(* PLC project marvel_fem, Institute of Astronomy Onto 0.0.1 *)
(* stored: creationDateTime 2025-01-01T00:00:00.0, modificationDateTime 2025-01-01T00:00:00.0 *)

TYPE FemTemperaturesParts : STRUCT
  {attribute 'TcHmiSymbol.Show'}
  basePlate : SimpleTemperature;  (* FEM base plate temperature in °C *)
  {attribute 'TcHmiSymbol.Show'}
  electronics : SimpleTemperature;  (* FEM base plate temperature in °C *)
  {attribute 'TcHmiSymbol.Show'}
  ambient : SimpleTemperature;  (* FEM base plate temperature in °C *)
  {attribute 'TcHmiSymbol.Show'}
  fork : SimpleTemperature;  (* Telescope fork temperature in °C *)
  {attribute 'TcHmiSymbol.Show'}
  truss : SimpleTemperature;  (* Telescope truss temperature in °C *)
  {attribute 'TcHmiSymbol.Show'}
  spider : SimpleTemperature;  (* Telescope spider temperature in °C *)
  {attribute 'TcHmiSymbol.Show'}
  m1Cell : SimpleTemperature;  (* Telescope m1 cell temperature in °C *)
  {attribute 'TcHmiSymbol.Show'}
  spare : SimpleTemperature;  (* Telescope spare temperature in °C *)
END_STRUCT;
END_TYPE

TYPE FemParts : STRUCT
  {attribute 'TcHmiSymbol.Show'}
  fs : MTS50Axis;  (* The fibre selector stage *)
  {attribute 'TcHmiSymbol.Show'}
  cm : MTS50Axis;  (* The calibration mirror stage *)
  {attribute 'TcHmiSymbol.Show'}
  adc1 : ELL14Stage;  (* The ADC rotation 1 stage *)
  {attribute 'TcHmiSymbol.Show'}
  adc2 : ELL14Stage;  (* The ADC rotation 2 stage *)
  {attribute 'TcHmiSymbol.Show'}
  temp : FemTemperatures;  (* Temperatures measured by the front end *)
  {attribute 'TcHmiSymbol.Show'}
  relayGuideCam : SimpleRelay;  (* Relay to power on/off the guiding camera *)
  {attribute 'TcHmiSymbol.Show'}
  relayAcqCam : SimpleRelay;  (* Relay to power on/off the acquisition camera *)
  {attribute 'TcHmiSymbol.Show'}
  relayAdc : SimpleRelay;  (* Relay to power on/off both ADC controllers *)
  {attribute 'TcHmiSymbol.Show'}
  relayTT : SimpleRelay;  (* Relay to power on/off the Tip Tilt piezo driver *)
  {attribute 'TcHmiSymbol.Show'}
  ledHGF : Led;  (* HGF LED *)
  {attribute 'TcHmiSymbol.Show'}
  ledHSF : Led;  (* HSF LED *)
  {attribute 'TcHmiSymbol.Show'}
  ledUGF : Led;  (* UGF LED *)
  {attribute 'TcHmiSymbol.Show'}
  ledUSF : Led;  (* USF LED *)
  {attribute 'TcHmiSymbol.Show'}
  guideCam : GigECamera;  (* Guiding camera *)
  {attribute 'TcHmiSymbol.Show'}
  fvCam : GigECamera;  (* Fibre View camera *)
END_STRUCT;
END_TYPE

TYPE FemProcesses : STRUCT
  {attribute 'TcHmiSymbol.Show'}
  initialize : Process;  (* Start initializing the FEM *)
END_STRUCT;
END_TYPE

TYPE FemTemperaturesStatuses : STRUCT
  {attribute 'OPC.UA.DA' := '1'}
  {attribute 'OPC.UA.DA.Access' := '1'}
  {attribute 'TcHmiSymbol.Show'}
  health : HealthStatus;  (* Are all temperatures OK? *)
END_STRUCT;
END_TYPE

TYPE FemStatuses : STRUCT
  {attribute 'OPC.UA.DA' := '1'}
  {attribute 'OPC.UA.DA.Access' := '1'}
  {attribute 'TcHmiSymbol.Show'}
  init : InitializationStatus;
  {attribute 'OPC.UA.DA' := '1'}
  {attribute 'OPC.UA.DA.Access' := '1'}
  {attribute 'TcHmiSymbol.Show'}
  health : HealthStatus;
  {attribute 'OPC.UA.DA' := '1'}
  {attribute 'OPC.UA.DA.Access' := '1'}
  {attribute 'TcHmiSymbol.Show'}
  busy : BusyStatus;
END_STRUCT;
END_TYPE

TYPE FemConfig : STRUCT
  {attribute 'TcHmiSymbol.Show'}
  fsSim : BOOL;  (* TRUE if the fibre selector axis is simulated *)
  {attribute 'TcHmiSymbol.Show'}
  cmSim : BOOL;  (* TRUE if the calibration mirror motor is simulated *)
  {attribute 'TcHmiSymbol.Show'}
  adc1Sim : BOOL;  (* TRUE if the ADC stage 1 is simulated *)
  {attribute 'TcHmiSymbol.Show'}
  adc2Sim : BOOL;  (* TRUE if the ADC stage 2 is simulated *)
  {attribute 'TcHmiSymbol.Show'}
  psSim : BOOL;  (* TRUE if the 10V and 5V power supplies are simulated *)
  {attribute 'TcHmiSymbol.Show'}
  temp : FemTempConfig;  (* Temperatures config *)
END_STRUCT;
END_TYPE

TYPE FemTempConfig : STRUCT
  {attribute 'TcHmiSymbol.Show'}
  basePlate : MeasurementConfig;  (* FEM base plate config in °C *)
  {attribute 'TcHmiSymbol.Show'}
  electronics : MeasurementConfig;  (* FEM base plate config in °C *)
  {attribute 'TcHmiSymbol.Show'}
  ambient : MeasurementConfig;  (* FEM base plate config in °C *)
  {attribute 'TcHmiSymbol.Show'}
  fork : MeasurementConfig;  (* Telescope fork config in °C *)
  {attribute 'TcHmiSymbol.Show'}
  truss : MeasurementConfig;  (* Telescope truss config in °C *)
  {attribute 'TcHmiSymbol.Show'}
  spider : MeasurementConfig;  (* Telescope spider config in °C *)
  {attribute 'TcHmiSymbol.Show'}
  m1Cell : MeasurementConfig;  (* Telescope m1 cell config in °C *)
  {attribute 'TcHmiSymbol.Show'}
  spare : MeasurementConfig;  (* Telescope spare config in °C *)
END_STRUCT;
END_TYPE

TYPE M_SM_FemTemperatures : STRUCT
  {attribute 'OPC.UA.DA' := '1'}
  {attribute 'OPC.UA.DA.Access' := '1'}
  {attribute 'TcHmiSymbol.Show'}
  actualStatus : STRING;
  {attribute 'OPC.UA.DA' := '1'}
  {attribute 'TcHmiSymbol.Show'}
  stat : FemTemperaturesStatuses;
  {attribute 'OPC.UA.DA' := '1'}
  {attribute 'TcHmiSymbol.Show'}
  parts : M_SM_FemTemperaturesParts;
END_STRUCT;
END_TYPE

TYPE M_SM_Fem : STRUCT
  {attribute 'OPC.UA.DA' := '1'}
  {attribute 'OPC.UA.DA.Access' := '1'}
  {attribute 'TcHmiSymbol.Show'}
  actualStatus : STRING;
  {attribute 'OPC.UA.DA' := '1'}
  {attribute 'OPC.UA.DA.Access' := '1'}
  {attribute 'TcHmiSymbol.Show'}
  power5VOK : BOOL;
  {attribute 'OPC.UA.DA' := '1'}
  {attribute 'OPC.UA.DA.Access' := '1'}
  {attribute 'TcHmiSymbol.Show'}
  power5VOverload : BOOL;
  {attribute 'OPC.UA.DA' := '1'}
  {attribute 'OPC.UA.DA.Access' := '1'}
  {attribute 'TcHmiSymbol.Show'}
  power10VOK : BOOL;
  {attribute 'OPC.UA.DA' := '1'}
  {attribute 'OPC.UA.DA.Access' := '1'}
  {attribute 'TcHmiSymbol.Show'}
  power10VOverload : BOOL;
  {attribute 'OPC.UA.DA' := '1'}
  {attribute 'TcHmiSymbol.Show'}
  stat : FemStatuses;
  {attribute 'OPC.UA.DA' := '1'}
  {attribute 'TcHmiSymbol.Show'}
  parts : M_SM_FemParts;
  {attribute 'OPC.UA.DA' := '1'}
  {attribute 'TcHmiSymbol.Show'}
  proc : M_SM_FemProcesses;
END_STRUCT;
END_TYPE

TYPE M_SM_FemTemperaturesParts : STRUCT
  {attribute 'TcHmiSymbol.Show'}
  basePlate : M_SimpleTemperature;
  {attribute 'TcHmiSymbol.Show'}
  electronics : M_SimpleTemperature;
  {attribute 'TcHmiSymbol.Show'}
  ambient : M_SimpleTemperature;
  {attribute 'TcHmiSymbol.Show'}
  fork : M_SimpleTemperature;
  {attribute 'TcHmiSymbol.Show'}
  truss : M_SimpleTemperature;
  {attribute 'TcHmiSymbol.Show'}
  spider : M_SimpleTemperature;
  {attribute 'TcHmiSymbol.Show'}
  m1Cell : M_SimpleTemperature;
  {attribute 'TcHmiSymbol.Show'}
  spare : M_SimpleTemperature;
END_STRUCT;
END_TYPE

TYPE M_SM_FemParts : STRUCT
  {attribute 'TcHmiSymbol.Show'}
  fs : M_MTS50Axis;
  {attribute 'TcHmiSymbol.Show'}
  cm : M_MTS50Axis;
  {attribute 'TcHmiSymbol.Show'}
  adc1 : M_ELL14Stage;
  {attribute 'TcHmiSymbol.Show'}
  adc2 : M_ELL14Stage;
  {attribute 'TcHmiSymbol.Show'}
  temp : M_FemTemperatures;
  {attribute 'TcHmiSymbol.Show'}
  relayGuideCam : M_SimpleRelay;
  {attribute 'TcHmiSymbol.Show'}
  relayAcqCam : M_SimpleRelay;
  {attribute 'TcHmiSymbol.Show'}
  relayAdc : M_SimpleRelay;
  {attribute 'TcHmiSymbol.Show'}
  relayTT : M_SimpleRelay;
  {attribute 'TcHmiSymbol.Show'}
  ledHGF : M_Led;
  {attribute 'TcHmiSymbol.Show'}
  ledHSF : M_Led;
  {attribute 'TcHmiSymbol.Show'}
  ledUGF : M_Led;
  {attribute 'TcHmiSymbol.Show'}
  ledUSF : M_Led;
  {attribute 'TcHmiSymbol.Show'}
  guideCam : M_GigECamera;
  {attribute 'TcHmiSymbol.Show'}
  fvCam : M_GigECamera;
END_STRUCT;
END_TYPE

TYPE M_SM_FemProcesses : STRUCT
  {attribute 'TcHmiSymbol.Show'}
  initialize : M_Process;
END_STRUCT;
END_TYPE

FUNCTION_BLOCK SM_FemTemperatures
  VAR_OUTPUT
    {attribute 'OPC.UA.DA' := '1'}
    {attribute 'OPC.UA.DA.Access' := '1'}
    actualStatus : STRING(30);  (* Current status description *)
    {attribute 'OPC.UA.DA' := '1'}
    stat : FemTemperaturesStatuses;  (* Statuses of the state machine *)
    {attribute 'OPC.UA.DA' := '1'}
    parts : FemTemperaturesParts;  (* Parts of the state machine *)
  END_VAR
  VAR_IN_OUT
    {attribute 'OPC.UA.DA' := '0'}
    config_ref : FemTempConfig;  (* Active configuration of the FEM temperatures *)
  END_VAR

            parts.basePlate( config := config_ref.basePlate );
parts.electronics( config := config_ref.electronics );
parts.ambient( config := config_ref.ambient );
parts.fork( config := config_ref.fork );
parts.truss( config := config_ref.truss );
parts.spider( config := config_ref.spider );
parts.m1Cell( config := config_ref.m1Cell );
parts.spare( config := config_ref.spare );
stat.health := F_HealthStatus(
    superState := TRUE,
    isGood := ((NOT(parts.basePlate.stat.health = HealthStatus.bad)) OR (parts.basePlate.stat.enabled = EnabledStatus.disabled)) AND (((NOT(parts.electronics.stat.health = HealthStatus.bad)) OR (parts.electronics.stat.enabled = EnabledStatus.disabled)) AND (((NOT(parts.ambient.stat.health = HealthStatus.bad)) OR (parts.ambient.stat.enabled = EnabledStatus.disabled)) AND (((NOT(parts.fork.stat.health = HealthStatus.bad)) OR (parts.fork.stat.enabled = EnabledStatus.disabled)) AND (((NOT(parts.truss.stat.health = HealthStatus.bad)) OR (parts.truss.stat.enabled = EnabledStatus.disabled)) AND (((NOT(parts.spider.stat.health = HealthStatus.bad)) OR (parts.spider.stat.enabled = EnabledStatus.disabled)) AND (((NOT(parts.m1Cell.stat.health = HealthStatus.bad)) OR (parts.m1Cell.stat.enabled = EnabledStatus.disabled)) AND ((NOT(parts.spare.stat.health = HealthStatus.bad)) OR (parts.spare.stat.enabled = EnabledStatus.disabled)))))))),
    hasWarning := (parts.basePlate.stat.health = HealthStatus.warning) OR ((parts.electronics.stat.health = HealthStatus.warning) OR ((parts.ambient.stat.health = HealthStatus.warning) OR ((parts.fork.stat.health = HealthStatus.warning) OR ((parts.truss.stat.health = HealthStatus.warning) OR ((parts.spider.stat.health = HealthStatus.warning) OR ((parts.m1Cell.stat.health = HealthStatus.warning) OR (parts.spare.stat.health = HealthStatus.warning))))))));

          

METHOD _copyFromModel_SM_FemTemperatures
  VAR_IN_OUT
    {attribute 'OPC.UA.DA' := '0'}
    model : M_SM_FemTemperatures;
  END_VAR
                  THIS^.parts.basePlate._copyFromModel_SimpleTemperature( model := model.parts.basePlate );
THIS^.parts.electronics._copyFromModel_SimpleTemperature( model := model.parts.electronics );
THIS^.parts.ambient._copyFromModel_SimpleTemperature( model := model.parts.ambient );
THIS^.parts.fork._copyFromModel_SimpleTemperature( model := model.parts.fork );
THIS^.parts.truss._copyFromModel_SimpleTemperature( model := model.parts.truss );
THIS^.parts.spider._copyFromModel_SimpleTemperature( model := model.parts.spider );
THIS^.parts.m1Cell._copyFromModel_SimpleTemperature( model := model.parts.m1Cell );
THIS^.parts.spare._copyFromModel_SimpleTemperature( model := model.parts.spare );

                
END_METHOD

METHOD _copyToModel_SM_FemTemperatures
  VAR_IN_OUT
    {attribute 'OPC.UA.DA' := '0'}
    model : M_SM_FemTemperatures;
  END_VAR
                  model.actualStatus := THIS^.actualStatus;
model.stat := THIS^.stat;
THIS^.parts.basePlate._copyToModel_SimpleTemperature( model := model.parts.basePlate );
THIS^.parts.electronics._copyToModel_SimpleTemperature( model := model.parts.electronics );
THIS^.parts.ambient._copyToModel_SimpleTemperature( model := model.parts.ambient );
THIS^.parts.fork._copyToModel_SimpleTemperature( model := model.parts.fork );
THIS^.parts.truss._copyToModel_SimpleTemperature( model := model.parts.truss );
THIS^.parts.spider._copyToModel_SimpleTemperature( model := model.parts.spider );
THIS^.parts.m1Cell._copyToModel_SimpleTemperature( model := model.parts.m1Cell );
THIS^.parts.spare._copyToModel_SimpleTemperature( model := model.parts.spare );

                
END_METHOD
END_FUNCTION_BLOCK

FUNCTION_BLOCK SM_Fem
  VAR_OUTPUT
    {attribute 'OPC.UA.DA' := '1'}
    {attribute 'OPC.UA.DA.Access' := '1'}
    actualStatus : STRING(30);  (* Current status description *)
    {attribute 'OPC.UA.DA' := '1'}
    {attribute 'OPC.UA.DA.Access' := '1'}
    power5VOK AT %I* : BOOL;  (* 5V power supply is OK *)
    {attribute 'OPC.UA.DA' := '1'}
    {attribute 'OPC.UA.DA.Access' := '1'}
    power5VOverload AT %I* : BOOL;  (* 5V power supply is overloaded *)
    {attribute 'OPC.UA.DA' := '1'}
    {attribute 'OPC.UA.DA.Access' := '1'}
    power10VOK AT %I* : BOOL;  (* 10V power supply is OK *)
    {attribute 'OPC.UA.DA' := '1'}
    {attribute 'OPC.UA.DA.Access' := '1'}
    power10VOverload AT %I* : BOOL;  (* 10V power supply is overloaded *)
    {attribute 'OPC.UA.DA' := '1'}
    stat : FemStatuses;  (* Statuses of the state machine *)
    {attribute 'OPC.UA.DA' := '1'}
    parts : FemParts;  (* Parts of the state machine *)
    {attribute 'OPC.UA.DA' := '1'}
    proc : FemProcesses;  (* Processes of the state machine *)
  END_VAR
  VAR_IN_OUT
    {attribute 'OPC.UA.DA' := '0'}
    number : USINT;  (* Number of the unit (1-4) *)
    {attribute 'OPC.UA.DA' := '0'}
    operator_ref : OperatorStatus;  (* Reference to the operator (observer/tech) *)
    {attribute 'OPC.UA.DA' := '0'}
    activity_ref : ActivityStatus;  (* Shared activity status *)
    {attribute 'OPC.UA.DA' := '0'}
    services_ref : Services;  (* Shared services *)
    {attribute 'OPC.UA.DA' := '0'}
    config_ref : FemConfig;  (* Active configuration of the FEM *)
  END_VAR

            parts.fs(
    isEnabled := (NOT(stat.init = InitializationStatus.locked)) AND (operator_ref = OperatorStatus.tech),
    usePosLimitSwitch := TRUE,
    useNegLimitSwitch := TRUE,
    invertPosLimitSwitch := TRUE,
    invertNegLimitSwitch := TRUE);
parts.cm(
    isEnabled := (NOT(stat.init = InitializationStatus.locked)) AND (operator_ref = OperatorStatus.tech),
    usePosLimitSwitch := TRUE,
    useNegLimitSwitch := TRUE,
    invertPosLimitSwitch := TRUE,
    invertNegLimitSwitch := TRUE);
parts.adc1(
    isEnabled := (NOT(stat.init = InitializationStatus.locked)) AND (operator_ref = OperatorStatus.tech),
    simulated := config_ref.adc1Sim);
parts.adc2(
    isEnabled := (NOT(stat.init = InitializationStatus.locked)) AND (operator_ref = OperatorStatus.tech),
    simulated := config_ref.adc2Sim);
parts.temp( config_ref := config_ref.temp );
parts.relayGuideCam( isEnabled := (NOT(stat.init = InitializationStatus.locked)) AND (operator_ref = OperatorStatus.tech) );
parts.relayAcqCam( isEnabled := (NOT(stat.init = InitializationStatus.locked)) AND (operator_ref = OperatorStatus.tech) );
parts.relayAdc( isEnabled := (NOT(stat.init = InitializationStatus.locked)) AND (operator_ref = OperatorStatus.tech) );
parts.relayTT( isEnabled := (NOT(stat.init = InitializationStatus.locked)) AND (operator_ref = OperatorStatus.tech) );
parts.ledHGF( isEnabled := (NOT(stat.init = InitializationStatus.locked)) AND (operator_ref = OperatorStatus.tech) );
parts.ledHSF( isEnabled := (NOT(stat.init = InitializationStatus.locked)) AND (operator_ref = OperatorStatus.tech) );
parts.ledUGF( isEnabled := (NOT(stat.init = InitializationStatus.locked)) AND (operator_ref = OperatorStatus.tech) );
parts.ledUSF( isEnabled := (NOT(stat.init = InitializationStatus.locked)) AND (operator_ref = OperatorStatus.tech) );
parts.guideCam();
parts.fvCam();
stat.health := F_HealthStatus(
    superState := NOT(stat.init = InitializationStatus.shutdown),
    isGood := (NOT(stat.init = InitializationStatus.initializingFailed)) AND (power5VOK AND (power10VOK AND (((parts.fs.stat.health = HealthStatus.good) OR (parts.fs.stat.health = HealthStatus.warning)) AND (((parts.cm.stat.health = HealthStatus.good) OR (parts.cm.stat.health = HealthStatus.warning)) AND (((parts.temp.stat.health = HealthStatus.good) OR (parts.temp.stat.health = HealthStatus.warning)) AND (((parts.adc1.stat.health = HealthStatus.good) OR (parts.adc1.stat.health = HealthStatus.warning)) AND (((parts.adc2.stat.health = HealthStatus.good) OR (parts.adc2.stat.health = HealthStatus.warning)) AND (((parts.guideCam.stat.health = HealthStatus.good) OR (parts.guideCam.stat.health = HealthStatus.warning)) AND ((parts.fvCam.stat.health = HealthStatus.good) OR (parts.fvCam.stat.health = HealthStatus.warning)))))))))),
    hasWarning := (parts.fs.stat.health = HealthStatus.warning) OR ((parts.cm.stat.health = HealthStatus.warning) OR ((parts.temp.stat.health = HealthStatus.warning) OR ((parts.adc1.stat.health = HealthStatus.warning) OR ((parts.adc2.stat.health = HealthStatus.warning) OR ((parts.guideCam.stat.health = HealthStatus.warning) OR (parts.fvCam.stat.health = HealthStatus.warning)))))));
stat.busy := F_BusyStatus(
    superState := NOT(stat.init = InitializationStatus.shutdown),
    isBusy := (parts.fs.stat.busy = BusyStatus.busy) OR ((parts.cm.stat.busy = BusyStatus.busy) OR ((parts.adc1.stat.busy = BusyStatus.busy) OR ((parts.adc2.stat.busy = BusyStatus.busy) OR ((parts.relayGuideCam.stat.busy = BusyStatus.busy) OR ((parts.relayAcqCam.stat.busy = BusyStatus.busy) OR ((parts.relayAdc.stat.busy = BusyStatus.busy) OR ((parts.relayTT.stat.busy = BusyStatus.busy) OR ((parts.ledHGF.stat.busy = BusyStatus.busy) OR ((parts.ledHSF.stat.busy = BusyStatus.busy) OR ((parts.ledUGF.stat.busy = BusyStatus.busy) OR ((parts.ledUSF.stat.busy = BusyStatus.busy) OR ((parts.guideCam.stat.busy = BusyStatus.busy) OR (parts.fvCam.stat.busy = BusyStatus.busy))))))))))))));
proc.initialize( isEnabled := NOT(stat.init = InitializationStatus.initializing) );

          

METHOD _copyFromModel_SM_Fem
  VAR_IN_OUT
    {attribute 'OPC.UA.DA' := '0'}
    model : M_SM_Fem;
  END_VAR
                  THIS^.parts.fs._copyFromModel_MTS50Axis( model := model.parts.fs );
THIS^.parts.cm._copyFromModel_MTS50Axis( model := model.parts.cm );
THIS^.parts.adc1._copyFromModel_ELL14Stage( model := model.parts.adc1 );
THIS^.parts.adc2._copyFromModel_ELL14Stage( model := model.parts.adc2 );
THIS^.parts.temp._copyFromModel_FemTemperatures( model := model.parts.temp );
THIS^.parts.relayGuideCam._copyFromModel_SimpleRelay( model := model.parts.relayGuideCam );
THIS^.parts.relayAcqCam._copyFromModel_SimpleRelay( model := model.parts.relayAcqCam );
THIS^.parts.relayAdc._copyFromModel_SimpleRelay( model := model.parts.relayAdc );
THIS^.parts.relayTT._copyFromModel_SimpleRelay( model := model.parts.relayTT );
THIS^.parts.ledHGF._copyFromModel_Led( model := model.parts.ledHGF );
THIS^.parts.ledHSF._copyFromModel_Led( model := model.parts.ledHSF );
THIS^.parts.ledUGF._copyFromModel_Led( model := model.parts.ledUGF );
THIS^.parts.ledUSF._copyFromModel_Led( model := model.parts.ledUSF );
THIS^.parts.guideCam._copyFromModel_GigECamera( model := model.parts.guideCam );
THIS^.parts.fvCam._copyFromModel_GigECamera( model := model.parts.fvCam );
THIS^.proc.initialize._copyFromModel_Process( model := model.proc.initialize );

                
END_METHOD

METHOD _copyToModel_SM_Fem
  VAR_IN_OUT
    {attribute 'OPC.UA.DA' := '0'}
    model : M_SM_Fem;
  END_VAR
                  model.actualStatus := THIS^.actualStatus;
model.power5VOK := THIS^.power5VOK;
model.power5VOverload := THIS^.power5VOverload;
model.power10VOK := THIS^.power10VOK;
model.power10VOverload := THIS^.power10VOverload;
model.stat := THIS^.stat;
THIS^.parts.fs._copyToModel_MTS50Axis( model := model.parts.fs );
THIS^.parts.cm._copyToModel_MTS50Axis( model := model.parts.cm );
THIS^.parts.adc1._copyToModel_ELL14Stage( model := model.parts.adc1 );
THIS^.parts.adc2._copyToModel_ELL14Stage( model := model.parts.adc2 );
THIS^.parts.temp._copyToModel_FemTemperatures( model := model.parts.temp );
THIS^.parts.relayGuideCam._copyToModel_SimpleRelay( model := model.parts.relayGuideCam );
THIS^.parts.relayAcqCam._copyToModel_SimpleRelay( model := model.parts.relayAcqCam );
THIS^.parts.relayAdc._copyToModel_SimpleRelay( model := model.parts.relayAdc );
THIS^.parts.relayTT._copyToModel_SimpleRelay( model := model.parts.relayTT );
THIS^.parts.ledHGF._copyToModel_Led( model := model.parts.ledHGF );
THIS^.parts.ledHSF._copyToModel_Led( model := model.parts.ledHSF );
THIS^.parts.ledUGF._copyToModel_Led( model := model.parts.ledUGF );
THIS^.parts.ledUSF._copyToModel_Led( model := model.parts.ledUSF );
THIS^.parts.guideCam._copyToModel_GigECamera( model := model.parts.guideCam );
THIS^.parts.fvCam._copyToModel_GigECamera( model := model.parts.fvCam );
THIS^.proc.initialize._copyToModel_Process( model := model.proc.initialize );

                
END_METHOD
END_FUNCTION_BLOCK
